% RSLogix 500 project Presure Digital Control.RSS, saved by version 8.30.00.16 %
PROJECT "UNTITLED"    % processor: Bul.1763 MicroLogix 1100 Series B %

PROGRAM FILES
  LAD 2 "MAIN"  3 rungs
  LAD 3 "DIGITAL IO"  5 rungs
  LAD 4 "CONTROLS"  9 rungs

DATA FILES
  O0 OUTPUT  4 elements
  I1 INPUT  6 elements
  S2 STATUS  66 elements
  B3 BINARY  4 elements
  T4 TIMER  3 elements
  C5 COUNTER  1 elements
  R6 CONTROL  1 elements
  N7 INTEGER  1 elements
  F8 FLOAT  1 elements

LADDER 2 "MAIN"
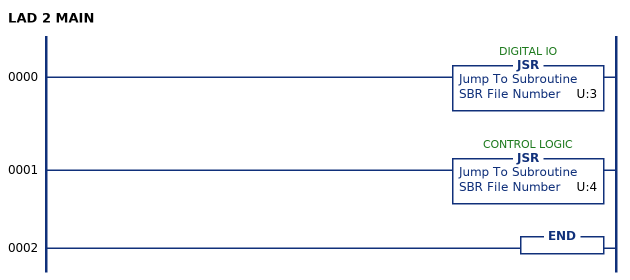
% Rung: 0 %
SOR JSR U:3 EOR
%   U:3  "DIGITAL IO" %
% Rung: 1 %
SOR JSR U:4 EOR
%   U:4  "CONTROL LOGIC" %
% Rung: 2 %
SOR END EOR

LADDER 3 "DIGITAL IO"
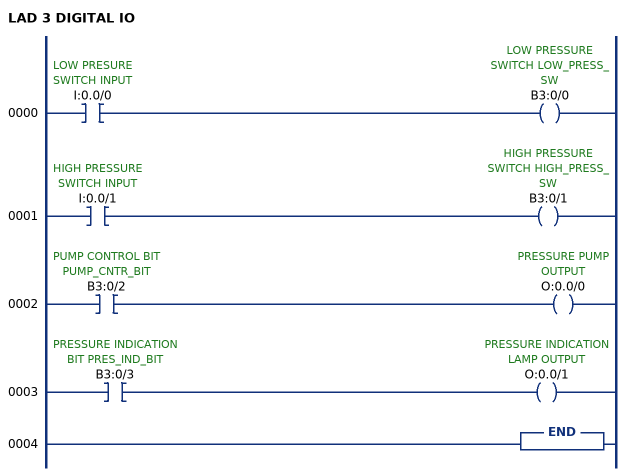
% Rung: 0 %
SOR XIC I:0.0/0 OTE B3:0/0 EOR
%   I:0.0/0  "LOW PRESURE SWITCH INPUT" %
%   B3:0/0  LOW_PRESS_SW  "LOW PRESSURE SWITCH" %
% Rung: 1 %
SOR XIC I:0.0/1 OTE B3:0/1 EOR
%   I:0.0/1  "HIGH PRESSURE SWITCH INPUT" %
%   B3:0/1  HIGH_PRESS_SW  "HIGH PRESSURE SWITCH" %
% Rung: 2 %
SOR XIC B3:0/2 OTE O:0.0/0 EOR
%   B3:0/2  PUMP_CNTR_BIT  "PUMP CONTROL BIT" %
%   O:0.0/0  "PRESSURE PUMP OUTPUT" %
% Rung: 3 %
SOR XIC B3:0/3 OTE O:0.0/1 EOR
%   B3:0/3  PRES_IND_BIT  "PRESSURE INDICATION BIT" %
%   O:0.0/1  "PRESSURE INDICATION LAMP OUTPUT" %
% Rung: 4 %
SOR END EOR

LADDER 4 "CONTROLS"
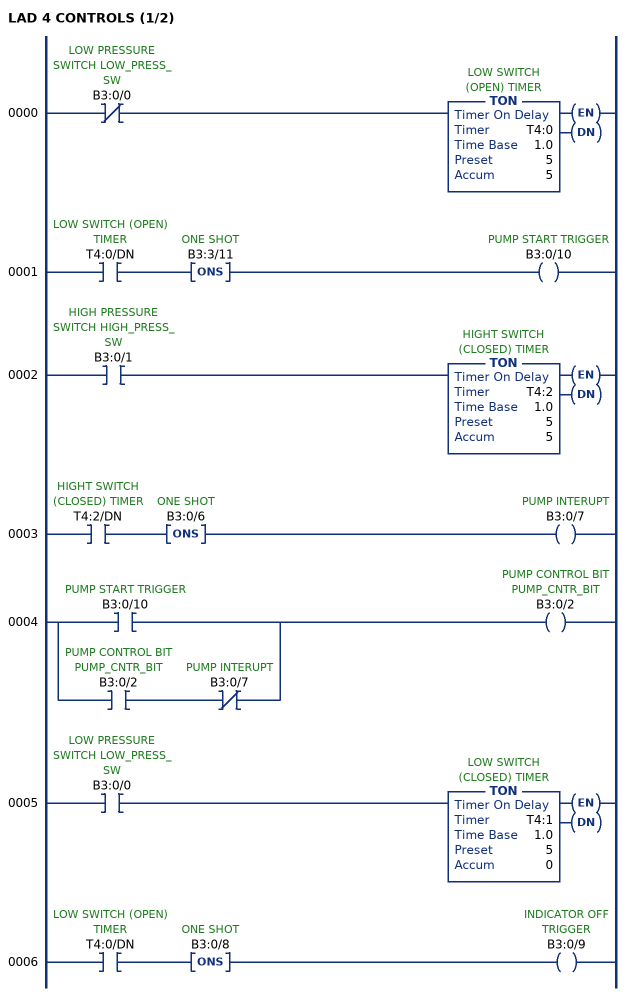
% Rung: 0 %
SOR XIO B3:0/0 TON T4:0 1.0 5 5 EOR
%   B3:0/0  LOW_PRESS_SW  "LOW PRESSURE SWITCH" %
%   T4:0  "LOW SWITCH (OPEN) TIMER" %
% Rung: 1 %
SOR XIC T4:0/DN ONS B3:3/11 OTE B3:0/10 EOR
%   T4:0  "LOW SWITCH (OPEN) TIMER" %
%   B3:3/11  "ONE SHOT" %
%   B3:0/10  "PUMP START TRIGGER" %
% Rung: 2 %
SOR XIC B3:0/1 TON T4:2 1.0 5 5 EOR
%   B3:0/1  HIGH_PRESS_SW  "HIGH PRESSURE SWITCH" %
%   T4:2  "HIGHT SWITCH (CLOSED) TIMER" %
% Rung: 3 %
SOR XIC T4:2/DN ONS B3:0/6 OTE B3:0/7 EOR
%   T4:2  "HIGHT SWITCH (CLOSED) TIMER" %
%   B3:0/6  "ONE SHOT" %
%   B3:0/7  "PUMP INTERUPT" %
% Rung: 4 %
SOR BST XIC B3:0/10 NXB XIC B3:0/2 XIO B3:0/7 BND OTE B3:0/2 EOR
%   B3:0/10  "PUMP START TRIGGER" %
%   B3:0/2  PUMP_CNTR_BIT  "PUMP CONTROL BIT" %
%   B3:0/7  "PUMP INTERUPT" %
% Rung: 5 %
SOR XIC B3:0/0 TON T4:1 1.0 5 0 EOR
%   B3:0/0  LOW_PRESS_SW  "LOW PRESSURE SWITCH" %
%   T4:1  "LOW SWITCH (CLOSED) TIMER" %
% Rung: 6 %
SOR XIC T4:0/DN ONS B3:0/8 OTE B3:0/9 EOR
%   T4:0  "LOW SWITCH (OPEN) TIMER" %
%   B3:0/8  "ONE SHOT" %
%   B3:0/9  "INDICATOR OFF TRIGGER" %

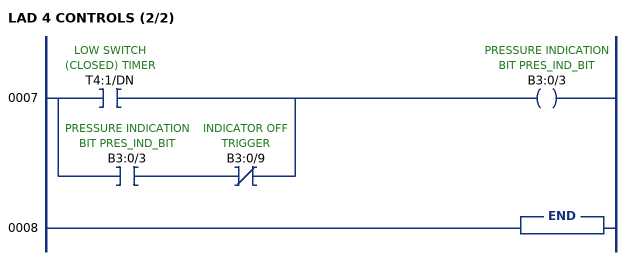
% Rung: 7 %
SOR BST XIC T4:1/DN NXB XIC B3:0/3 XIO B3:0/9 BND OTE B3:0/3 EOR
%   T4:1  "LOW SWITCH (CLOSED) TIMER" %
%   B3:0/3  PRES_IND_BIT  "PRESSURE INDICATION BIT" %
%   B3:0/9  "INDICATOR OFF TRIGGER" %
% Rung: 8 %
SOR END EOR

OTHER DOCUMENTED ADDRESSES
  B3:0/4  "ONE SHOT"
  B3:0/5  "ONE SHOT"

DATA TABLE (non-zero values as saved)
DATA B3
% B3:0 % 0X0146 0X0000 0X0000 0X0000
DATA T4
% .PRE .ACC %
% T4:0 % 5 5
% T4:1 % 5 0
% T4:2 % 5 5
